RoboDK station: Simspons.rdk

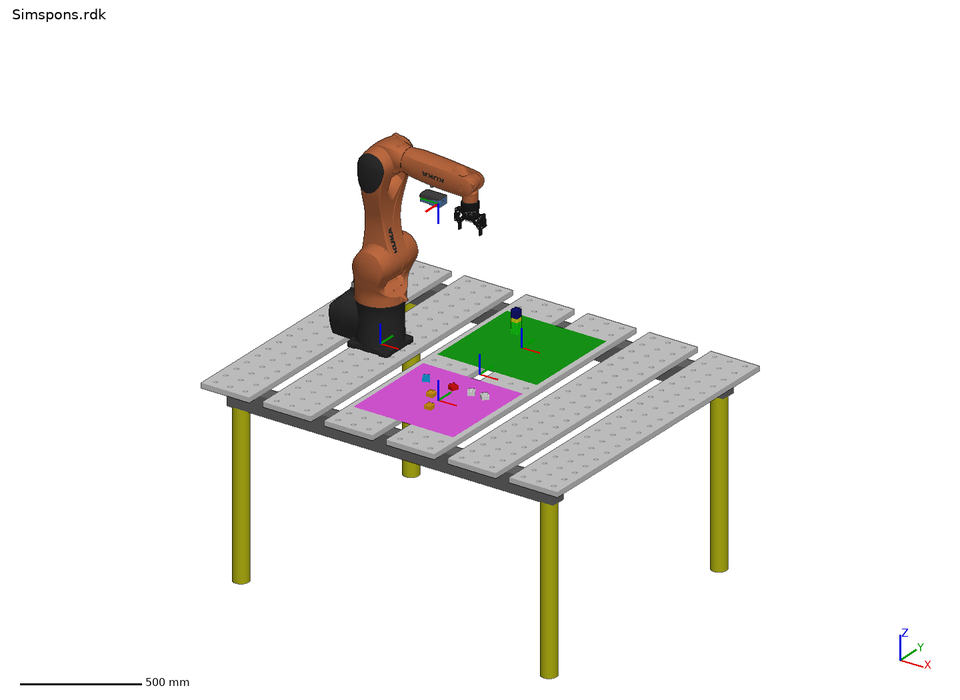
[picture v0: the station drawn from its stored meshes, robots at their saved joint values, targets as dots, program paths as lines]
Station Simspons. Poses are relative to the parent item; angles as X-Y-Z fixed-axis rotations.
  - frame KUKAFrame at (0, 1000, 0) mm
    - robot KUKA (model KUKA KR 6 R900 sixx): 6 axes, payload 6 kg, reach 901 mm, repeatability 0.03 mm, weight 52 kg
        modified DH rows (alpha deg, a mm, theta deg, d mm): 0, 0, 0, 400; -90, 25, 0, 0; 0, 455, -90, 0; -90, 35, 0, 420; 90, 0, 0, 0; -90, 0, 180, 80
        joint limits [-170, -190, -120, -185, -120, -350] to [170, 45, 156, 185, 120, 350]; home [0, -90, 90, 0, 0, 0]; saved at [0, -89.55, 93.632, -180, -85.918, 0]
      - tool Gripper, TCP at (0, 0, 130) mm, size 147.4 x 146.8 x 75 mm
  - frame World at (500, 1000, 0) mm
    - object Table at (0, 0, 0) mm, size 1790.7 x 1447.8 x 914.4 mm, geometry from welding_table.sld
    - frame Bricks at (0, -300, 1) mm
      - object Plane 1m x 1m at (0, 0, 0) mm, size 500 x 500 x 0.2 mm, geometry from plane_1m.sld
      - object Orange at (-30, 0, 0) mm, rotated rx 0 ry 0 rz 91 deg, size 31.7 x 31.7 x 23.7 mm, geometry from LEGO_DUPLO_BRICK_2X2.igs
      - object Orange at (0, -100, 0) mm, rotated rx 0 ry 0 rz 2 deg, size 31.7 x 31.7 x 23.7 mm, geometry from LEGO_DUPLO_BRICK_2X2.igs
      - object Red at (0, 100, 0) mm, rotated rx 0 ry 0 rz 70 deg, size 31.7 x 31.7 x 23.7 mm, geometry from LEGO_DUPLO_BRICK_2X2.igs
      - object White at (150, 100, 0) mm, rotated rx 0 ry 0 rz 50 deg, size 31.7 x 31.7 x 23.7 mm, geometry from LEGO_DUPLO_BRICK_2X2.igs
      - object White at (75, 100, 0) mm, rotated rx 0 ry 0 rz 28 deg, size 31.7 x 31.7 x 23.7 mm, geometry from LEGO_DUPLO_BRICK_2X2.igs
      - object Light_Blue at (-150, 100, 0) mm, rotated rx 0 ry 0 rz 33 deg, size 31.7 x 31.7 x 23.7 mm, geometry from LEGO_DUPLO_BRICK_2X2.igs
    - frame Assembly at (0, 300, 1) mm
      - object Plane 1m x 1m at (0, 0, 0) mm, size 500 x 500 x 0.2 mm, geometry from plane_1m.sld
      - object Light_Green at (-114.89, 83.69, 0) mm, rotated rx 0 ry 0 rz 1.25 deg, size 31.7 x 31.7 x 23.7 mm, geometry from LEGO_DUPLO_BRICK_2X2.igs
      - object Light_Green at (-84.13, 83.91, 18) mm, rotated rx 0 ry 0 rz 89.19 deg, size 31.7 x 31.7 x 23.7 mm, geometry from LEGO_DUPLO_BRICK_2X2.igs
      - object Light_Green at (-115.06, 83.77, 36) mm, rotated rx 0 ry 0 rz 1.08 deg, size 31.7 x 31.7 x 23.7 mm, geometry from LEGO_DUPLO_BRICK_2X2.igs
      - object Yellow at (-115.07, 84.03, 54) mm, rotated rx 0 ry 0 rz 0.89 deg, size 31.7 x 31.7 x 23.7 mm, geometry from LEGO_DUPLO_BRICK_2X2.igs
      - object Dark_Blue at (-115.65, 115.69, 72) mm, rotated rx 0 ry 0 rz -88.83 deg, size 31.7 x 31.7 x 23.7 mm, geometry from LEGO_DUPLO_BRICK_2X2.igs
      - object Dark_Blue at (-83.5, 84.34, 90) mm, rotated rx 0 ry 0 rz 90.39 deg, size 31.7 x 31.7 x 23.7 mm, geometry from LEGO_DUPLO_BRICK_2X2.igs
    - frame Camera at (0, -300, 900) mm, rotated rx 180 ry 0 rz -90 deg
      - object SICK VSPP-5f2113 at (0, 0, 0) mm, rotated rx 0 ry 0 rz -90 deg, size 53 x 116 x 38 mm, geometry from Cam2D_SICK_VSPP_5F2113.sld
  - program ReplaceBricks (1 instructions, listed below)

--- program ReplaceBricks (robot KUKA) ---
  Objekte ersetzen
